# EPICS autosave request: iocBoot/ioc13xps_test/auto_positions.req
file "CARS_motor_positions.req",         P=13xps3:, M=m1
~
